TYPE Timer :
STRUCT
	timerTime : TIME;
	timerStart : BOOL;
	timerCon : TON;
END_STRUCT
END_TYPE

(* stored: Version 1.1.0.1, ProductVersion 3.1.4024.12
   DUT Timer: Id {27d2dc1f-45fc-4ce0-8295-bfc49af49711} *)
